{attribute 'qualified_only'}
//{attribute 'strict'}
TYPE E_CAMERA_Name :
(
	CAM01		:= 1,
	CAM02		:= 2,
	CAM03		:= 3,
	CAM04		:= 4,
	CAM05		:= 5,
	CAM06		:= 6,
	CAM07		:= 7,
	CAM08		:= 8,
	CAM09		:= 9,
	CAM10		:= 10,
	CAM11		:= 11,
	CAM12		:= 12
);
END_TYPE

(* stored: Version 1.1.0.1
   DUT E_CAMERA_Name: Id {1cc37441-22ff-4e79-aa12-690a5aeb9f73} *)
